FUNCTION_BLOCK FB_DropSpeedComp

VAR_INPUT
  fMasterSpeed          : LREAL; //[m/s]
  fDropTravelDistance   : LREAL; //[m]
END_VAR

VAR_OUTPUT
  fDropPlacementError   : LREAL;
END_VAR

VAR
  _bEnable              : BOOL := TRUE;
  _fDropSpeed           : LREAL := fL_DropSpeed;                 // [m/s]
  _fDropSpeedDeadTime   : LREAL := fL_DropSpeedAddTime;          // [ms]
END_VAR

VAR CONSTANT
  fL_DropSpeed          : LREAL := 6;        // DropSpeed for start compensation
  fL_DropSpeedAddTime   : LREAL := 2.15;  //0.388889; // DropSpeed compensation, additional dead time [ms]
END_VAR

(*Speed compensation*)
IF _bEnable AND (_fDropSpeed > 0) THEN
	fDropPlacementError :=  (  (fDropTravelDistance / _fDropSpeed)
                        + (_fDropSpeedDeadTime / 1000))             (*[s]*)
                        * fMasterSpeed;
ELSE
  fDropPlacementError := 0;
END_IF;

PROPERTY bEnable : BOOL
GET
bEnable := _bEnable;
END_GET
SET
_bEnable := bEnable;
END_SET
END_PROPERTY

PROPERTY fDropSpeed : LREAL
GET
fDropSpeed := _fDropSpeed;
END_GET
SET
_fDropSpeed := fDropSpeed;
END_SET
END_PROPERTY

PROPERTY fDropSpeedDeadTime : LREAL
GET
fDropSpeedDeadTime := _fDropSpeedDeadTime;
END_GET
SET
_fDropSpeedDeadTime := fDropSpeedDeadTime;
END_SET
END_PROPERTY

END_FUNCTION_BLOCK

(* stored: Version 1.1.0.1, ProductVersion 3.1.4024.9
   POU FB_DropSpeedComp: Id {31156881-dc16-4df5-a26b-2bb900ace12f}, SpecialFunc None
   Property bEnable: Id {47387335-4acf-45af-94b0-c212f662bfbd}
   Get Get: Id {d3d8720f-d96a-487a-bfb8-ca90ae5694d5}
   Set Set: Id {af6f84f6-b1ba-4dc8-8cfa-ec1ee10dcd28}
   Property fDropSpeed: Id {2f104349-ca5b-4875-b549-8cf775b3f6e6}
   Get Get: Id {6d12ca1b-ae7a-4b3b-b098-ab0757cae63e}
   Set Set: Id {d8edc7f0-427f-43eb-adcc-183ede0e1a46}
   Property fDropSpeedDeadTime: Id {8380f83b-2ae2-4634-9b6e-e67dda41a57f}
   Get Get: Id {00f9ba1a-0ac5-4c6d-ad08-e3025cbdcb3c}
   Set Set: Id {cf8943c4-b9bb-491c-8050-2543558bba18} *)
